// TwinCAT 3 PLC project Sample02
// ProgramVersion: 3.1.4022.1
// libraries:
//   Tc2_Standard, * (Beckhoff Automation GmbH)
//   Tc2_System, * (Beckhoff Automation GmbH)
//   Tc3_Module, * (Beckhoff Automation GmbH)
// project tree:
//   GVLs/ Param.TcGVL (not stored)
//   / PlcTask.TcTTO (not stored)
//   POUs/ FB_Base.TcPOU, FB_Observer.TcPOU, FB_SubjectBase.TcPOU, FB_SubjectNew.TcPOU, MAIN.TcPOU, I_Observer.TcIO (not stored), I_Subject.TcIO (not stored)
// real-time tasks:
//   TASK PlcTask: cycle T#10ms, priority 20, ADS port 350

// ---- POUs/FB_Base.TcPOU
FUNCTION_BLOCK PUBLIC FB_Base
VAR_INPUT
END_VAR
VAR_OUTPUT
END_VAR
VAR
END_VAR

END_FUNCTION_BLOCK

// ---- POUs/FB_Observer.TcPOU
FUNCTION_BLOCK PUBLIC FB_Observer IMPLEMENTS I_Observer
VAR
	fValue				: LREAL;
END_VAR

PROPERTY PUBLIC fActualValue : LREAL
GET
fActualValue := THIS^.fValue;
END_GET
END_PROPERTY

METHOD PUBLIC Update
VAR_INPUT
	fValue			: LREAL;
END_VAR
THIS^.fValue := fValue;
END_METHOD

END_FUNCTION_BLOCK

// ---- POUs/FB_SubjectBase.TcPOU
FUNCTION_BLOCK PUBLIC FB_SubjectBase IMPLEMENTS I_Subject
VAR
	aObservers			: ARRAY [1..Param.cMaxObservers] OF I_Observer;
END_VAR

METHOD PUBLIC Attach : BOOL
VAR_INPUT
	ipObserver				: I_Observer;
END_VAR
VAR
	nIndex					: INT := 0;
END_VAR
Attach := FALSE;
IF (ipObserver = 0) THEN
	RETURN;
END_IF

// is the observer already registered?
FOR nIndex := 1 TO Param.cMaxObservers DO	
	IF (THIS^.aObservers[nIndex] = ipObserver) THEN
		RETURN;
	END_IF
END_FOR

// save the observer object into the array of observers and send the actual value
FOR nIndex := 1 TO Param.cMaxObservers DO
	IF (THIS^.aObservers[nIndex] = 0) THEN
		THIS^.aObservers[nIndex] := ipObserver;
		Attach := TRUE;
		EXIT;					
	END_IF
END_FOR
END_METHOD

METHOD PUBLIC Detach : BOOL
VAR_INPUT
	ipObserver		: I_Observer;
END_VAR
VAR
	nIndex			: INT := 0;
END_VAR
Detach := FALSE;
IF (ipObserver = 0) THEN
	RETURN;
END_IF

FOR nIndex := 1 TO Param.cMaxObservers DO
	IF (THIS^.aObservers[nIndex] = ipObserver) THEN
		THIS^.aObservers[nIndex] := 0;
		Detach := TRUE;	
	END_IF
END_FOR
END_METHOD

END_FUNCTION_BLOCK

// ---- POUs/FB_SubjectNew.TcPOU
FUNCTION_BLOCK PUBLIC FB_SubjectNew EXTENDS FB_Base IMPLEMENTS I_Subject
VAR
	fbDelay				: TON;
	fbDrand				: DRAND;
	fValue				: LREAL;
	fbSubjectBase		: FB_SubjectBase;
END_VAR

// creates every sec a random value and invoke the update method
fbDelay(IN := TRUE, PT := T#500MS);
IF (fbDelay.Q) THEN	
	fbDelay(IN := FALSE);
	fbDrand(SEED := TO_INT(ADR(fValue)));
	fValue := fbDrand.Num * 1.0;
	THIS^.Notify();
END_IF

METHOD PUBLIC Attach : BOOL
VAR_INPUT
	ipObserver				: I_Observer;
END_VAR
Attach := FALSE;
IF (THIS^.fbSubjectBase.Attach(ipObserver)) THEN
	ipObserver.Update(THIS^.fValue);
	Attach := TRUE;
END_IF
END_METHOD

METHOD PUBLIC Detach : BOOL
VAR_INPUT
	ipObserver		: I_Observer;
END_VAR
Detach := THIS^.fbSubjectBase.Detach(ipObserver);
END_METHOD

{attribute 'monitoring':='call'}
PROPERTY PUBLIC fActualValue : LREAL
GET
fActualValue := THIS^.fValue;
END_GET
END_PROPERTY

METHOD PRIVATE Notify
VAR	
	nIndex		: INT := 0;
END_VAR
FOR nIndex := 1 TO Param.cMaxObservers DO
	IF (THIS^.fbSubjectBase.aObservers[nIndex] <> 0) THEN
		THIS^.fbSubjectBase.aObservers[nIndex].Update(THIS^.fActualValue);
	END_IF
END_FOR
END_METHOD

END_FUNCTION_BLOCK

// ---- POUs/MAIN.TcPOU
PROGRAM MAIN
VAR
	fbSubject 			: FB_SubjectNew;
	fbObserver1 		: FB_Observer;
	fbObserver2 		: FB_Observer;
	
	bAttachObserver1	: BOOL;
	bAttachObserver2	: BOOL;

	bDetachObserver1	: BOOL;
	bDetachObserver2	: BOOL;
END_VAR

fbSubject();

IF (bAttachObserver1) THEN
	fbSubject.Attach(fbObserver1);
	bAttachObserver1 := FALSE;
END_IF

IF (bAttachObserver2) THEN
	fbSubject.Attach(fbObserver2);
	bAttachObserver2 := FALSE;
END_IF

IF (bDetachObserver1) THEN
	fbSubject.Detach(fbObserver1);
	bDetachObserver1 := FALSE;
END_IF

IF (bDetachObserver2) THEN
	fbSubject.Detach(fbObserver2);
	bDetachObserver2 := FALSE;
END_IF

END_PROGRAM
